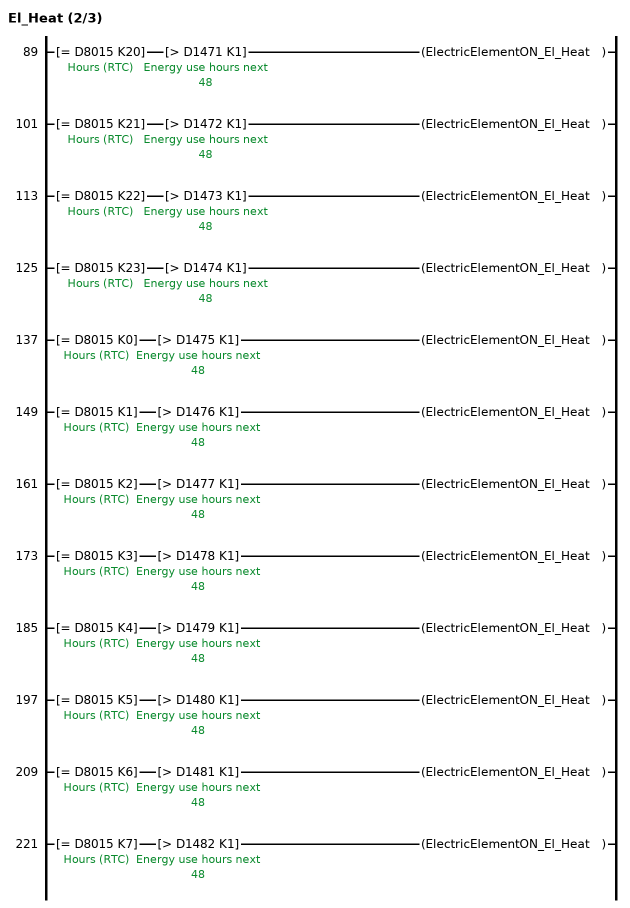
89    LD=     D8015 K20  ; Hours (RTC)
      AND>    D1471 K1  ; Energy use hours next 48
      OUT     ElectricElementON_El_Heat
        [note] 20,00
101   LD=     D8015 K21  ; Hours (RTC)
      AND>    D1472 K1  ; Energy use hours next 48
      OUT     ElectricElementON_El_Heat
        [note] 21,00
113   LD=     D8015 K22  ; Hours (RTC)
      AND>    D1473 K1  ; Energy use hours next 48
      OUT     ElectricElementON_El_Heat
        [note] 22,00
125   LD=     D8015 K23  ; Hours (RTC)
      AND>    D1474 K1  ; Energy use hours next 48
      OUT     ElectricElementON_El_Heat
        [note] 23,00
137   LD=     D8015 K0  ; Hours (RTC)
      AND>    D1475 K1  ; Energy use hours next 48
      OUT     ElectricElementON_El_Heat
        [note] 00,00
149   LD=     D8015 K1  ; Hours (RTC)
      AND>    D1476 K1  ; Energy use hours next 48
      OUT     ElectricElementON_El_Heat
        [note] 01,00
161   LD=     D8015 K2  ; Hours (RTC)
      AND>    D1477 K1  ; Energy use hours next 48
      OUT     ElectricElementON_El_Heat
        [note] 02,00
173   LD=     D8015 K3  ; Hours (RTC)
      AND>    D1478 K1  ; Energy use hours next 48
      OUT     ElectricElementON_El_Heat
        [note] 03,00
185   LD=     D8015 K4  ; Hours (RTC)
      AND>    D1479 K1  ; Energy use hours next 48
      OUT     ElectricElementON_El_Heat
        [note] 04,00
197   LD=     D8015 K5  ; Hours (RTC)
      AND>    D1480 K1  ; Energy use hours next 48
      OUT     ElectricElementON_El_Heat
        [note] 05,00
209   LD=     D8015 K6  ; Hours (RTC)
      AND>    D1481 K1  ; Energy use hours next 48
      OUT     ElectricElementON_El_Heat
        [note] 06,00
221   LD=     D8015 K7  ; Hours (RTC)
      AND>    D1482 K1  ; Energy use hours next 48
      OUT     ElectricElementON_El_Heat
        [note] 07,00
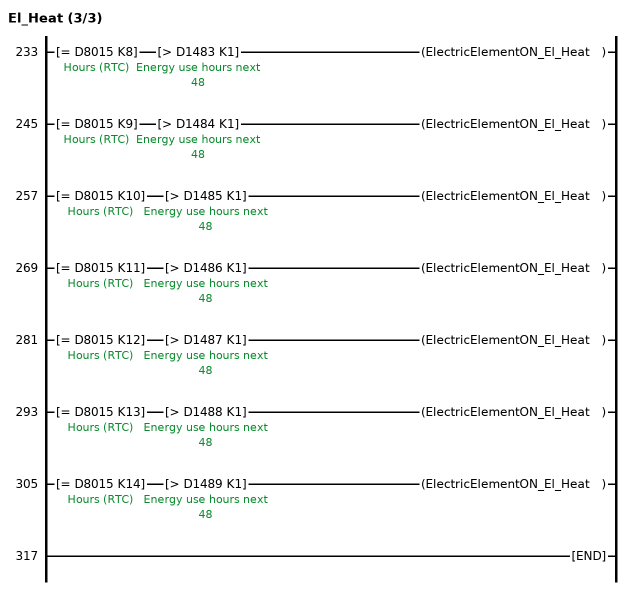
233   LD=     D8015 K8  ; Hours (RTC)
      AND>    D1483 K1  ; Energy use hours next 48
      OUT     ElectricElementON_El_Heat
        [note] 08,00
245   LD=     D8015 K9  ; Hours (RTC)
      AND>    D1484 K1  ; Energy use hours next 48
      OUT     ElectricElementON_El_Heat
        [note] 09,00
257   LD=     D8015 K10  ; Hours (RTC)
      AND>    D1485 K1  ; Energy use hours next 48
      OUT     ElectricElementON_El_Heat
        [note] 10,00
269   LD=     D8015 K11  ; Hours (RTC)
      AND>    D1486 K1  ; Energy use hours next 48
      OUT     ElectricElementON_El_Heat
        [note] 11,00
281   LD=     D8015 K12  ; Hours (RTC)
      AND>    D1487 K1  ; Energy use hours next 48
      OUT     ElectricElementON_El_Heat
        [note] 12,00
293   LD=     D8015 K13  ; Hours (RTC)
      AND>    D1488 K1  ; Energy use hours next 48
      OUT     ElectricElementON_El_Heat
        [note] 13,00
305   LD=     D8015 K14  ; Hours (RTC)
      AND>    D1489 K1  ; Energy use hours next 48
      OUT     ElectricElementON_El_Heat
        [note] 14,00
317   END
END_PROGRAM

PROGRAM Sol_Heat
VAR
  TempDiffPer1C : DINT;  (* Temerature differents pes 1 C *)
  TempShift : DINT;  (* Temperature shift *)
  Ring2ShiftAdd : DINT;
  Ring2ShiftAdded : DINT;
  TempDiff : DINT;  (* Heat Graph temp difference *)
  BaseTemp : INT;  (* Base temperatuere for calc *)
  SetValue : INT;  (* Value from Graph *)
  Ring2Interval : TIMER;  (* Ring 1 actuator valve update interval *)
  TempdifferentsforPID : INT;  (* Temp different for PID *)
  TempInc : INT;  (* Temperature increment to actuator *)
  Ring1Interval : TIMER;  (* Ring 1 actuator valve update interval *)
  changeable : BOOL;  (* temperatuure need correctsion *)
  TempdifferentsforPIDcor : DINT;  (* Corrected actuator value change *)
  Canadd : BOOL;  (* Can add more value *)
  CanTadd : BOOL;  (* Cant add more val *)
  changeable2 : BOOL;
  Solid_Heat_ON : BOOL;  (* Solid heater is activ mode *)
END_VAR
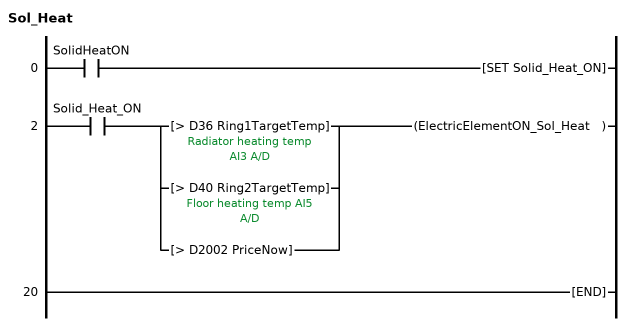
0     LD      SolidHeatON
      SET     Solid_Heat_ON
2     LD      Solid_Heat_ON
      LD>     D36 Ring1TargetTemp  ; Radiator heating temp AI3 A/D
      OR>     D40 Ring2TargetTemp  ; Floor heating temp AI5 A/D
      OR>     D2002 PriceNow
      ANB
      OUT     ElectricElementON_Sol_Heat
20    END
END_PROGRAM

PROGRAM Pum_Heat
VAR
  TempDiffPer1C : DINT;  (* Temerature differents pes 1 C *)
  TempShift : DINT;  (* Temperature shift *)
  Ring2ShiftAdd : DINT;
  Ring2ShiftAdded : DINT;
  TempDiff : DINT;  (* Heat Graph temp difference *)
  BaseTemp : INT;  (* Base temperatuere for calc *)
  SetValue : INT;  (* Value from Graph *)
  Ring2Interval : TIMER;  (* Ring 1 actuator valve update interval *)
  TempdifferentsforPID : INT;  (* Temp different for PID *)
  TempInc : INT;  (* Temperature increment to actuator *)
  Ring1Interval : TIMER;  (* Ring 1 actuator valve update interval *)
  changeable : BOOL;  (* temperatuure need correctsion *)
  TempdifferentsforPIDcor : DINT;  (* Corrected actuator value change *)
  Canadd : BOOL;  (* Can add more value *)
  CanTadd : BOOL;  (* Cant add more val *)
  changeable2 : BOOL;
  Pump_Heat_ON : BOOL;  (* Het pump funcsion is activ mode *)
END_VAR
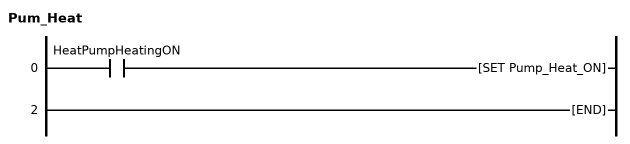
0     LD      HeatPumpHeatingON
      SET     Pump_Heat_ON
2     END
END_PROGRAM

PROGRAM PriceNow
VAR
  TempDiffPer1C : DINT;  (* Temerature differents pes 1 C *)
  TempShift : DINT;  (* Temperature shift *)
  Ring2ShiftAdd : DINT;
  Ring2ShiftAdded : DINT;
  TempDiff : DINT;  (* Heat Graph temp difference *)
  BaseTemp : INT;  (* Base temperatuere for calc *)
  SetValue : INT;  (* Value from Graph *)
  Ring2Interval : TIMER;  (* Ring 1 actuator valve update interval *)
  TempdifferentsforPID : INT;  (* Temp different for PID *)
  TempInc : INT;  (* Temperature increment to actuator *)
  Ring1Interval : TIMER;  (* Ring 1 actuator valve update interval *)
  changeable : BOOL;  (* temperatuure need correctsion *)
  TempdifferentsforPIDcor : DINT;  (* Corrected actuator value change *)
  Canadd : BOOL;  (* Can add more value *)
  CanTadd : BOOL;  (* Cant add more val *)
  changeable2 : BOOL;
  Solid_Heat_ON : BOOL;  (* Solid heater is activ mode *)
END_VAR
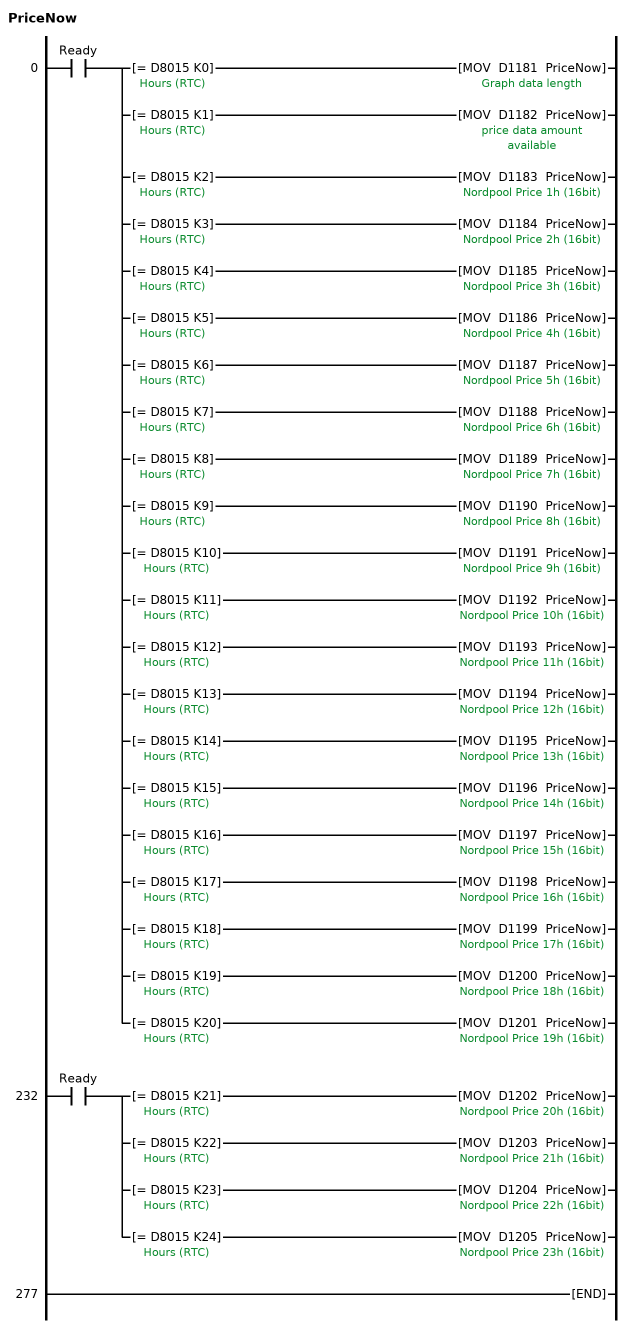
0     LD      Ready
      MPS
      AND=    D8015 K0  ; Hours (RTC)
      MOV     D1181 PriceNow  ; Graph data length
      MRD
      AND=    D8015 K1  ; Hours (RTC)
      MOV     D1182 PriceNow  ; price data amount available
      MRD
      AND=    D8015 K2  ; Hours (RTC)
      MOV     D1183 PriceNow  ; Nordpool Price 1h (16bit)
      MRD
      AND=    D8015 K3  ; Hours (RTC)
      MOV     D1184 PriceNow  ; Nordpool Price 2h (16bit)
      MRD
      AND=    D8015 K4  ; Hours (RTC)
      MOV     D1185 PriceNow  ; Nordpool Price 3h (16bit)
      MRD
      AND=    D8015 K5  ; Hours (RTC)
      MOV     D1186 PriceNow  ; Nordpool Price 4h (16bit)
      MRD
      AND=    D8015 K6  ; Hours (RTC)
      MOV     D1187 PriceNow  ; Nordpool Price 5h (16bit)
      MRD
      AND=    D8015 K7  ; Hours (RTC)
      MOV     D1188 PriceNow  ; Nordpool Price 6h (16bit)
      MRD
      AND=    D8015 K8  ; Hours (RTC)
      MOV     D1189 PriceNow  ; Nordpool Price 7h (16bit)
      MRD
      AND=    D8015 K9  ; Hours (RTC)
      MOV     D1190 PriceNow  ; Nordpool Price 8h (16bit)
      MRD
      AND=    D8015 K10  ; Hours (RTC)
      MOV     D1191 PriceNow  ; Nordpool Price 9h (16bit)
      MRD
      AND=    D8015 K11  ; Hours (RTC)
      MOV     D1192 PriceNow  ; Nordpool Price 10h (16bit)
      MRD
      AND=    D8015 K12  ; Hours (RTC)
      MOV     D1193 PriceNow  ; Nordpool Price 11h (16bit)
      MRD
      AND=    D8015 K13  ; Hours (RTC)
      MOV     D1194 PriceNow  ; Nordpool Price 12h (16bit)
      MRD
      AND=    D8015 K14  ; Hours (RTC)
      MOV     D1195 PriceNow  ; Nordpool Price 13h (16bit)
      MRD
      AND=    D8015 K15  ; Hours (RTC)
      MOV     D1196 PriceNow  ; Nordpool Price 14h (16bit)
      MRD
      AND=    D8015 K16  ; Hours (RTC)
      MOV     D1197 PriceNow  ; Nordpool Price 15h (16bit)
      MRD
      AND=    D8015 K17  ; Hours (RTC)
      MOV     D1198 PriceNow  ; Nordpool Price 16h (16bit)
      MRD
      AND=    D8015 K18  ; Hours (RTC)
      MOV     D1199 PriceNow  ; Nordpool Price 17h (16bit)
      MRD
      AND=    D8015 K19  ; Hours (RTC)
      MOV     D1200 PriceNow  ; Nordpool Price 18h (16bit)
      MPP
      AND=    D8015 K20  ; Hours (RTC)
      MOV     D1201 PriceNow  ; Nordpool Price 19h (16bit)
232   LD      Ready
      MPS
      AND=    D8015 K21  ; Hours (RTC)
      MOV     D1202 PriceNow  ; Nordpool Price 20h (16bit)
      MRD
      AND=    D8015 K22  ; Hours (RTC)
      MOV     D1203 PriceNow  ; Nordpool Price 21h (16bit)
      MRD
      AND=    D8015 K23  ; Hours (RTC)
      MOV     D1204 PriceNow  ; Nordpool Price 22h (16bit)
      MPP
      AND=    D8015 K24  ; Hours (RTC)
      MOV     D1205 PriceNow  ; Nordpool Price 23h (16bit)
277   END
END_PROGRAM

// device comments not shown above
M1  ; EMG button act.
M30  ; Prognose download
M36  ; PrognoseButton
D58  ; Ring1TargetTemp
D68  ; HeatFlowLiters
D70  ; Target temp floor heat
D72  ; Tank energy capacity *100
D1850  ; NextDayAvrTemp
D1852  ; NextDayAvrWind
D1854  ; NextDayAvrClody
D1874  ; Building area
D2004  ; Energy Price Now
D2006  ; TankWaterCapacity
D2008  ; Day energy use
D2010  ; Energy consumption yesterday
D2012  ; HetedEnergyInLastH
D2014  ; El.Heating element power
D2020  ; Real time heating
M67  ; Nextday to Today
M69  ; Data is updateted
M70  ; Sort Data
Y005  ; Domestic water circ Pump
D22  ; DA2 (0..4000 10V)
D50  ; AI40 A/D
D52  ; AI41 A/D
D54  ; AI12 A/D
D60  ; Modbus_stack
D1036  ; Domestic water max
D1038  ; Domestic water min
D1040  ; Heating graph max
D1042  ; Heating graph min
D1044  ; Radiator  graph max
D1046  ; Radiator  graph min
D1069  ; Nordpool Data Error
D1180  ; Today or yesterday
D1233  ; Nordpool Price 51h (16bit)
D1298  ; Sort data cylce
D1540  ; January day length
D1541  ; February day length
D1542  ; March day length
D1543  ; April day length
D1544  ; May day length
D1545  ; Jun day length
D1546  ; Jul day length
D1554  ; radiant flux Max
D1600  ; W20-.. .; 0-200W
D1601  ; W16-19; 0-200W
D1602  ; W12-15 0-200W
D1603  ; W8- 11  0-200W
D1604  ; W4-7     0-200W
D1605  ; W0-3   0-200W
D1606  ; W20-.. .; 201-400W
D1607  ; W16-19; - 201-400W
D1608  ; W12-15 -  201-400W
D1609  ; W8- 11 - 201-400W
D1610  ; W4-7 - 201-400W
D1611  ; W0-3 - 201-400W
D1612  ; W20-.. .; - 401-600W
D1613  ; W16-19; - 401-600W
D1614  ; W12-15 - 401-600W
D1615  ; W8- 11 - 401-600W
D1616  ; W4-7 - 401-600W
D1617  ; W0-3  - 401-600W
D1618  ; W20-.. .; - 601-800W
D1619  ; W16-19; 601-800W
D1620  ; W12-15 601-800W
D1621  ; W8- 11  601-800W
D1622  ; W4-7   601-800W
D1623  ; W0-3   601-800W
D1624  ; W20-.. .; - 801-1000W
D1625  ; W16-19; 801-1000W
D1626  ; W12-15 801-1000W
D1627  ; W8- 11  801-1000W
D1628  ; W4-7   801-1000W
D1629  ; W0-3   801-1000W
D1630  ; W20-.. .; - 1001-1200W
D1631  ; W16-19; 1001-1200W
D1632  ; W12-15 1001-1200W
D1633  ; W8- 11  1001-1200W
D1634  ; W4-7   1001-1200W
D1635  ; W0-3   1001-1200W
D1636  ; W20-.. .; - 1201-1500W
D1637  ; W16-19; 1201-1500W
D1638  ; W12-15 1201-1500W
D1639  ; W8- 11  1201-1500W
D1640  ; W4-7   1201-1500W
D1641  ; W0-3   1201-1500W
D1754  ; Weather Data (Wind) 3
D1755  ; Weather Data (Wind) 6
D1756  ; Weather Data (Wind) 9
D1757  ; Weather Data (Wind) 12
D1758  ; Weather Data (Wind) 15
D1759  ; Weather Data (Wind) 18
D1760  ; Weather Data (Wind) 21
D1761  ; Weather Data (Wind) 24
D1762  ; Weather Data (Wind) 27
D1763  ; Weather Data (Wind) 30
D1764  ; Weather Data (Wind) 33
D1765  ; Weather Data (Wind) 36
D1766  ; Weather Data (Wind) 39
D1767  ; Weather Data (Wind) 42
D1768  ; Weather Data (Wind) 45
D1769  ; Weather Data (Wind) 48
D1770  ; Weather Data (Wind) 51
D1771  ; Weather Data (Wind) 54
D1772  ; Weather Data (Wind) 57
D1773  ; Weather Data (Wind) 60
D1774  ; Weather Data (Wind) 63
D1775  ; Weather Data (Wind) 66
D1776  ; Weather Data (Wind) 69
D1777  ; Weather Data (Wind) 71
D1778  ; Weather Data (Wind) 73
D1779  ; Weather Data (Wind) 75
D1780  ; Weather Data (Wind) 78
D1781  ; Weather Data (Wind) 81
D1782  ; Weather Data (Wind) 84
D1783  ; Weather Data (Wind) 85
D1784  ; Weather Data (Wind) 88
D1785  ; Weather Data (Wind) 91
D1786  ; Weather Data (Wind) 94
D1787  ; Weather Data (Wind) 97
D1788  ; Weather Data (Wind) 100
D1789  ; Weather Data (Wind) 103
D1790  ; Weather Data (Wind) 106
D1791  ; Weather Data (Wind) 109
D1792  ; Weather Data (Wind) 102
D1793  ; Weather Data (Wind) 105
D1794  ; Weather Data (Wind) 108
D1795  ; Weather Data (Wind) 111
D1861  ; Tallinn
D1862  ; Ida-Virumaa
D1863  ; Kuressaare
D1864  ; Haapsalu
D1865  ; Paide
D1866  ; Pärnu
D1867  ; Tartu
D1868  ; Valga
D1870  ; Floor  graph max
D1872  ; Floor  graph max
